// TIA Portal project "IndustrialDemoController" (V15.1)

(* hardware
DEVICE "S7-1200 station_1"  S7-1200 Station
   slot 0: "Rack_0"  S7-1200 Rack  Rack  V1.0
   slot 1: "PLC_1"  CPU 1215C DC/DC/DC  6ES7 215-1AG40-0XB0  V4.1
*)

// ===== PLC "PLC_1"  CPU 1215C DC/DC/DC =====

VAR_GLOBAL   // PLC tag table "Default tag table"
   "Output0" AT %Q0.0 : Bool;
   "Output1" AT %Q0.1 : Bool;
   "Output2" AT %Q0.2 : Bool;
   "Output3" AT %Q0.3 : Bool;
   "Output4" AT %Q0.4 : Bool;
   "Output5" AT %Q0.5 : Bool;
   "Output6" AT %Q0.6 : Bool;
   "Output7" AT %Q0.7 : Bool;
   "Outputs" AT %QB0 : Byte;
END_VAR

DATA_BLOCK "ServerData"   // DB1
{ S7_Optimized_Access := 'FALSE' }
VERSION : 0.1
   VAR
      Outputs : Byte;
      In0 : Bool;
      In1 : Bool;
      In2 : Bool;
      In3 : Bool;
      In4 : Bool;
      In5 : Bool;
      In6 : Bool;
      In7 : Bool;
   END_VAR
BEGIN
END_DATA_BLOCK

ORGANIZATION_BLOCK "Main"   // OB1, LAD, ProgramCycle
TITLE = "Main Program Sweep (Cycle)"
{ S7_Optimized_Access := 'TRUE' }
VERSION : 0.1
   VAR_INPUT
      Initial_Call : Bool;   // Initial call of this OB
      Remanence : Bool;   // =True, if remanent data are available
   END_VAR
BEGIN

REGION Network 1
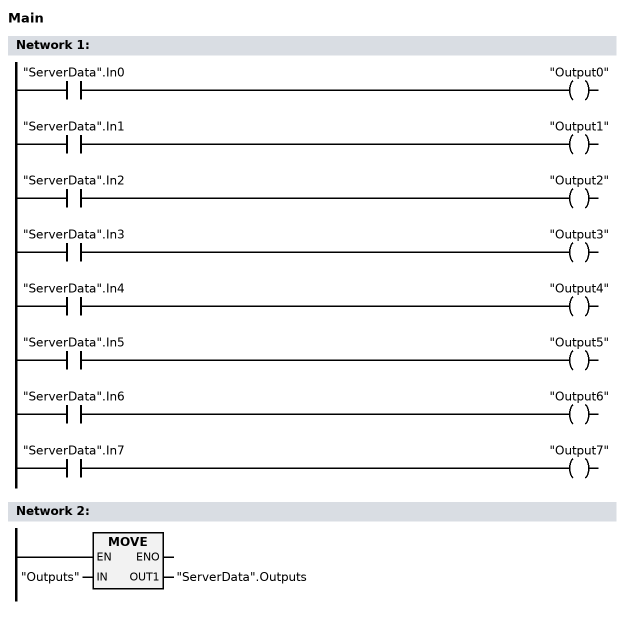
   RUNG wire#powerrail
      Contact( "ServerData".In0 )
      Coil( "Output0" )
   END_RUNG
   RUNG wire#powerrail
      Contact( "ServerData".In1 )
      Coil( "Output1" )
   END_RUNG
   RUNG wire#powerrail
      Contact( "ServerData".In2 )
      Coil( "Output2" )
   END_RUNG
   RUNG wire#powerrail
      Contact( "ServerData".In3 )
      Coil( "Output3" )
   END_RUNG
   RUNG wire#powerrail
      Contact( "ServerData".In4 )
      Coil( "Output4" )
   END_RUNG
   RUNG wire#powerrail
      Contact( "ServerData".In5 )
      Coil( "Output5" )
   END_RUNG
   RUNG wire#powerrail
      Contact( "ServerData".In6 )
      Coil( "Output6" )
   END_RUNG
   RUNG wire#powerrail
      Contact( "ServerData".In7 )
      Coil( "Output7" )
   END_RUNG
   // the same network as SCL:
   "Output0" := "ServerData".In0;
   "Output1" := "ServerData".In1;
   "Output2" := "ServerData".In2;
   "Output3" := "ServerData".In3;
   "Output4" := "ServerData".In4;
   "Output5" := "ServerData".In5;
   "Output6" := "ServerData".In6;
   "Output7" := "ServerData".In7;
END_REGION

REGION Network 2
   RUNG wire#powerrail
      Move(in := "Outputs", out1 => "ServerData".Outputs)
   END_RUNG
   // the same network as SCL:
   "ServerData".Outputs := "Outputs";
END_REGION
END_ORGANIZATION_BLOCK